{attribute 'qualified_only'}
{attribute 'strict'}
TYPE E_CutDirection :
(
    eCutX := 0,
    eCutY := 1
	//add other cutters here 
);
END_TYPE

(* stored: Version 1.1.0.1, ProductVersion 3.1.4024.15
   DUT E_CutDirection: Id {1bd624ee-db50-4079-b8fd-e0ddfc2065dc} *)
